// Mitsubishi GX Works2 project: Teaching   PLC: Q03UDV

PROGRAM MAIN
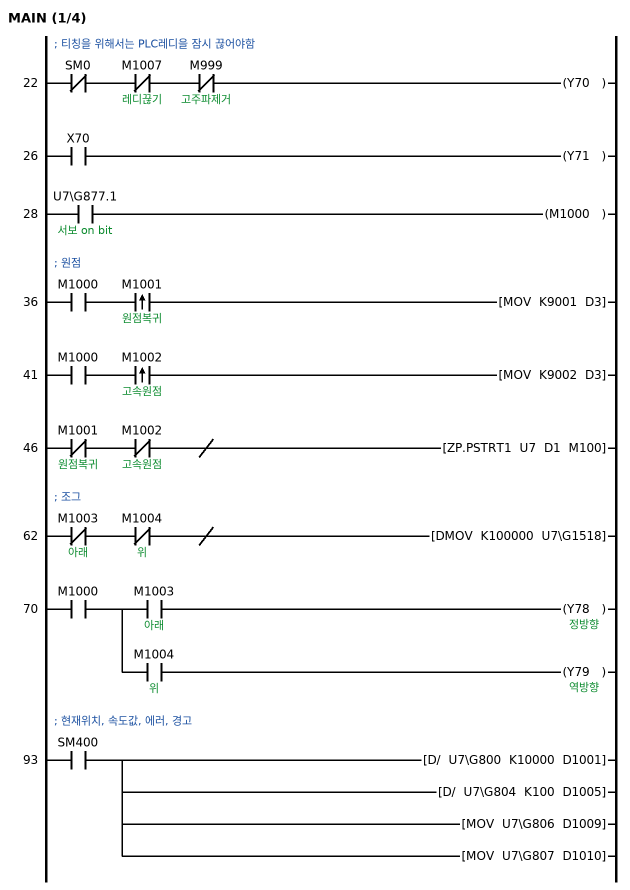
; 티칭을 위해서는 PLC레디을 잠시 끊어야함
22    LDI     SM0
      ANI     M1007  ; 레디끊기
      ANI     M999  ; 고주파제거
      OUT     Y70
26    LD      X70
      OUT     Y71
28    LD      U7\G877.1  ; 서보 on bit
      OUT     M1000
; 원점
36    LD      M1000
      ANDP    M1001  ; 원점복귀
      MOV     K9001 D3
41    LD      M1000
      ANDP    M1002  ; 고속원점
      MOV     K9002 D3
46    LDI     M1001  ; 원점복귀
      ANI     M1002  ; 고속원점
      INV
      ZP.PSTRT1 U7 D1 M100
; 조그
62    LDI     M1003  ; 아래
      ANI     M1004  ; 위
      INV
      DMOV    K100000 U7\G1518
70    LD      M1000
      MPS
      AND     M1003  ; 아래
      OUT     Y78  ; 정방향
      MPP
      AND     M1004  ; 위
      OUT     Y79  ; 역방향
; 현재위치, 속도값, 에러, 경고
93    LD      SM400
      D/      U7\G800 K10000 D1001
      D/      U7\G804 K100 D1005
      MOV     U7\G806 D1009
      MOV     U7\G807 D1010
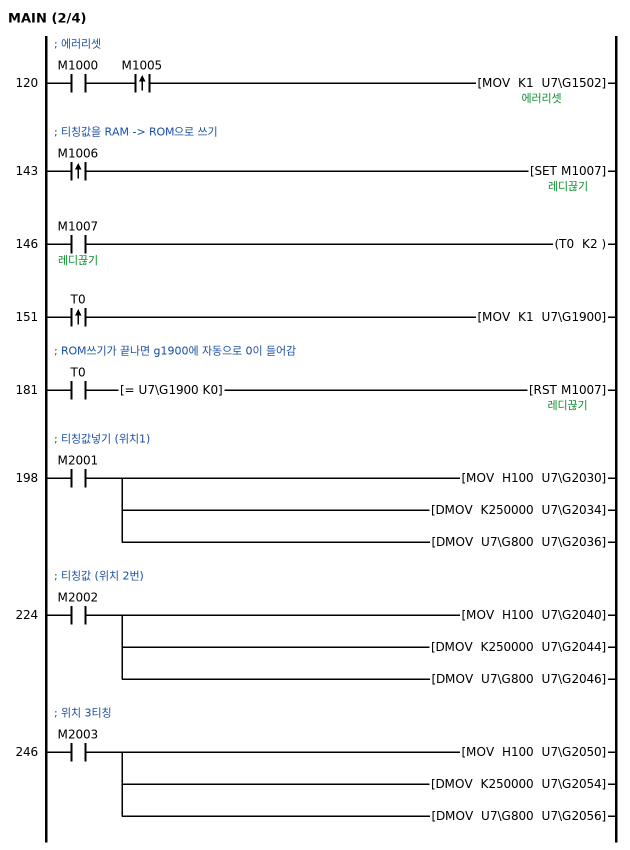
; 에러리셋
120   LD      M1000
      ANDP    M1005
      MOV     K1 U7\G1502  ; 에러리셋
; 티칭값을 RAM -> ROM으로 쓰기
143   LDP     M1006
      SET     M1007  ; 레디끊기
146   LD      M1007  ; 레디끊기
      OUT     T0 K2
151   LDP     T0
      MOV     K1 U7\G1900
; ROM쓰기가 끝나면 g1900에 자동으로 0이 들어감
181   LD      T0
      AND=    U7\G1900 K0
      RST     M1007  ; 레디끊기
; 티칭값넣기 (위치1)
198   LD      M2001
      MOV     H100 U7\G2030
      DMOV    K250000 U7\G2034
      DMOV    U7\G800 U7\G2036
; 티칭값 (위치 2번)
224   LD      M2002
      MOV     H100 U7\G2040
      DMOV    K250000 U7\G2044
      DMOV    U7\G800 U7\G2046
; 위치 3티칭
246   LD      M2003
      MOV     H100 U7\G2050
      DMOV    K250000 U7\G2054
      DMOV    U7\G800 U7\G2056
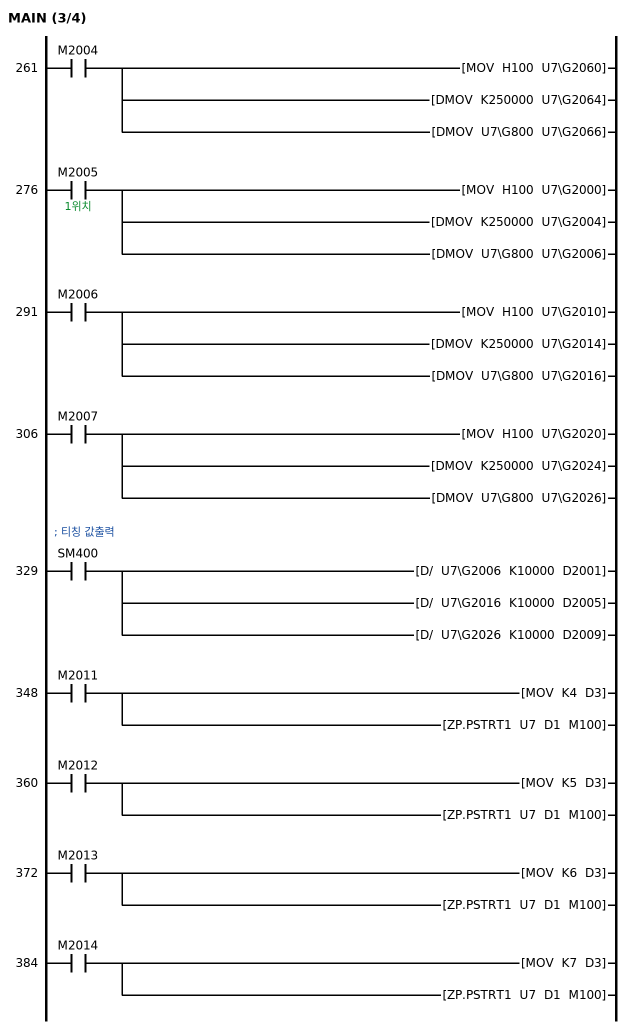
261   LD      M2004
      MOV     H100 U7\G2060
      DMOV    K250000 U7\G2064
      DMOV    U7\G800 U7\G2066
276   LD      M2005  ; 1위치
      MOV     H100 U7\G2000
      DMOV    K250000 U7\G2004
      DMOV    U7\G800 U7\G2006
291   LD      M2006
      MOV     H100 U7\G2010
      DMOV    K250000 U7\G2014
      DMOV    U7\G800 U7\G2016
306   LD      M2007
      MOV     H100 U7\G2020
      DMOV    K250000 U7\G2024
      DMOV    U7\G800 U7\G2026
; 티칭 값출력
329   LD      SM400
      D/      U7\G2006 K10000 D2001
      D/      U7\G2016 K10000 D2005
      D/      U7\G2026 K10000 D2009
348   LD      M2011
      MOV     K4 D3
      ZP.PSTRT1 U7 D1 M100
360   LD      M2012
      MOV     K5 D3
      ZP.PSTRT1 U7 D1 M100
372   LD      M2013
      MOV     K6 D3
      ZP.PSTRT1 U7 D1 M100
384   LD      M2014
      MOV     K7 D3
      ZP.PSTRT1 U7 D1 M100
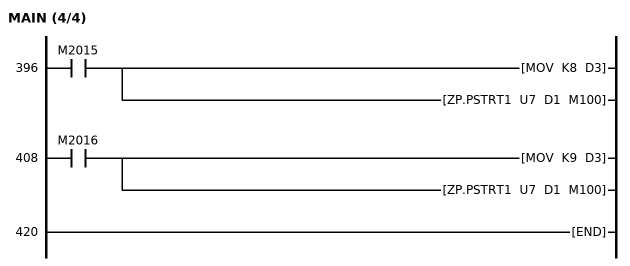
396   LD      M2015
      MOV     K8 D3
      ZP.PSTRT1 U7 D1 M100
408   LD      M2016
      MOV     K9 D3
      ZP.PSTRT1 U7 D1 M100
420   END
END_PROGRAM
